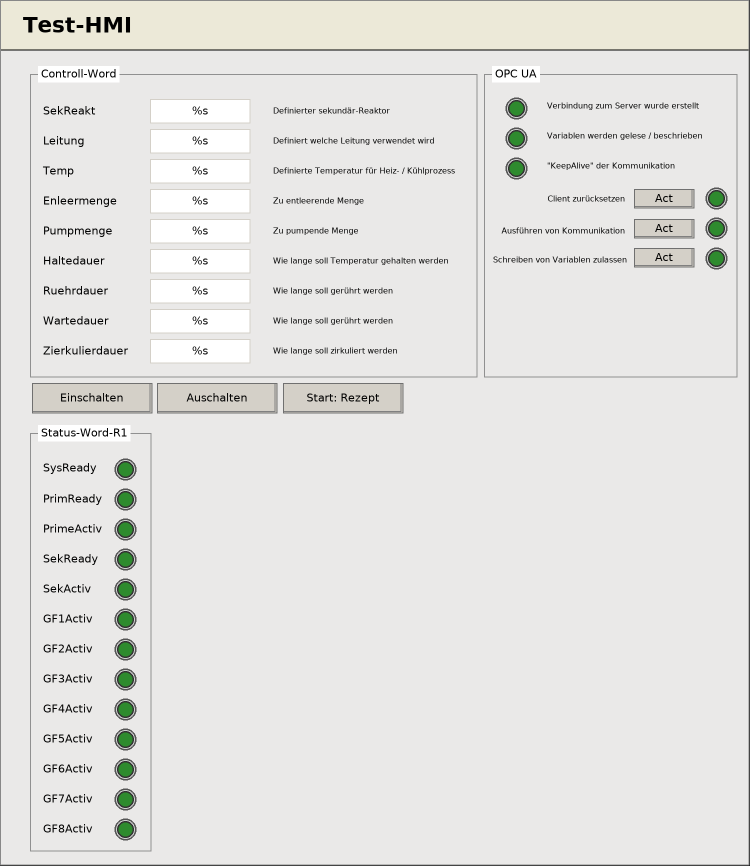
VISUALIZATION Test_Visu  // 750x866
    Rectangle (0,6 750x860)
    Rectangle (0,0 750x50)
    Label (20,0 480x50), "Test-HMI"
    GroupBox (30,66 447x311), "Controll-Word"
        Label (10,30 150x30), "SekReakt"
        Label (10,60 150x30), "Leitung"
        Label (10,90 150x30), "Temp"
        Label (10,120 150x30), "Enleermenge"
        Label (10,150 150x30), "Pumpmenge"
        Label (10,180 150x30), "Haltedauer"
        Label (10,210 150x30), "Ruehrdauer"
        Label (10,240 150x30), "Wartedauer"
        Label (10,270 150x30), "Zierkulierdauer"
        Textfield (120,33 100x24), "%s", text variable: GVL.Param_CW.SekReakt
            OnMouseClick: write GVL.Param_CW.SekReakt via Edit
        Textfield (120,63 100x24), "%s", text variable: GVL.Param_CW.Leitung
            OnMouseClick: write GVL.Param_CW.Leitung via Edit
        Textfield (120,93 100x24), "%s", text variable: GVL.Param_CW.Temp
            OnMouseClick: write GVL.Param_CW.Temp via Edit
        Textfield (120,123 100x24), "%s", text variable: GVL.Param_CW.Enlteermenge
            OnMouseClick: write GVL.Param_CW.Enlteermenge via Edit
        Textfield (120,153 100x24), "%s", text variable: GVL.Param_CW.Pumpmenge
            OnMouseClick: write GVL.Param_CW.Pumpmenge via Edit
        Textfield (120,183 100x24), "%s", text variable: GVL.Param_CW.Haltedauer
            OnMouseClick: write GVL.Param_CW.Haltedauer via Edit
        Textfield (120,213 100x24), "%s", text variable: GVL.Param_CW.Ruehrdauer
            OnMouseClick: write GVL.Param_CW.Ruehrdauer via Edit
        Textfield (120,243 100x24), "%s", text variable: GVL.Param_CW.Wartedauer
            OnMouseClick: write GVL.Param_CW.Wartedauer via Edit
        Textfield (120,273 100x24), "%s", text variable: GVL.Param_CW.Zirkulierdauer
            OnMouseClick: write GVL.Param_CW.Zirkulierdauer via Edit
        Label (240,30 300x30), "Definierter sekundär-Reaktor"
        Label (240,60 300x30), "Definiert welche Leitung verwendet wird"
        Label (240,90 300x30), "Definierte Temperatur für Heiz- / Kühlprozess"
        Label (240,120 300x30), "Zu entleerende Menge"
        Label (240,150 300x30), "Zu pumpende Menge"
        Label (240,180 300x30), "Wie lange soll Temperatur gehalten werden"
        Label (240,210 300x30), "Wie lange soll gerührt werden"
        Label (240,240 300x30), "Wie lange soll gerührt werden"
        Label (240,270 300x30), "Wie lange soll zirkuliert werden"
    GroupBox (30,425 121x426), "Status-Word-R1"
        Label (10,59 150x30), "PrimReady"
        Label (10,89 150x30), "PrimeActiv"
        Label (10,119 150x30), "SekReady"
        Label (10,149 150x30), "SekActiv"
        Label (10,179 150x30), "GF1Activ"
        Label (10,209 150x30), "GF2Activ"
        Label (10,239 150x30), "GF3Activ"
        Label (10,269 150x30), "GF4Activ"
        Label (10,299 150x30), "GF5Activ"
        Label (10,329 150x30), "GF6Activ"
        Label (10,359 150x30), "GF7Activ"
        Label (10,389 150x30), "GF8Activ"
        Lamp1 (83,62 25x25), variable: GVL_OPC_UA.SysSW_R1.GF8Activ, style: Lamp-Lamp1-Green
        Lamp1 (83,92 25x25), variable: GVL_OPC_UA.SysSW_R1.PrimActiv, style: Lamp-Lamp1-Green
        Lamp1 (83,122 25x25), variable: GVL_OPC_UA.SysSW_R1.SekReady, style: Lamp-Lamp1-Green
        Lamp1 (83,152 25x25), variable: GVL_OPC_UA.SysSW_R1.SekActiv, style: Lamp-Lamp1-Green
        Lamp1 (83,182 25x25), variable: GVL_OPC_UA.SysSW_R1.GF1Activ, style: Lamp-Lamp1-Green
        Lamp1 (83,212 25x25), variable: GVL_OPC_UA.SysSW_R1.GF2Activ, style: Lamp-Lamp1-Green
        Lamp1 (83,242 25x25), variable: GVL_OPC_UA.SysSW_R1.GF3Activ, style: Lamp-Lamp1-Green
        Lamp1 (83,272 25x25), variable: GVL_OPC_UA.SysSW_R1.GF4Activ, style: Lamp-Lamp1-Green
        Lamp1 (83,302 25x25), variable: GVL_OPC_UA.SysSW_R1.GF5Activ, style: Lamp-Lamp1-Green
        Lamp1 (83,332 25x25), variable: GVL_OPC_UA.SysSW_R1.GF6Activ, style: Lamp-Lamp1-Green
        Lamp1 (83,362 25x25), variable: GVL_OPC_UA.SysSW_R1.GF7Activ, style: Lamp-Lamp1-Green
        Lamp1 (83,392 25x25), variable: GVL_OPC_UA.SysSW_R1.GF8Activ, style: Lamp-Lamp1-Green
        Lamp1 (83,32 25x25), variable: GVL_OPC_UA.SysSW_R1.GF8Activ, style: Lamp-Lamp1-Green
    Button (283,383 120x30), "Start: Rezept"
        tap GVL.Start
    Button (32,383 120x30), "Einschalten"
        tap GVL.Start
        OnMouseClick: execute { Reaktoranlage.R1.M_M_ON(); }
    Button (157,383 120x30), "Auschalten"
        tap GVL.Start
        OnMouseClick: execute { Reaktoranlage.R1.M_M_OFF(); }
    GroupBox (484,66 253x311), "OPC UA"
        Lamp1 (20,30 25x25), variable: bWrite_Enable, style: Lamp-Lamp1-Green
        Lamp1 (20,60 25x25), variable: bReadBusy, style: Lamp-Lamp1-Green
        Lamp1 (20,90 25x25), variable: bKeepAlives, style: Lamp-Lamp1-Green
        Lamp1 (220,120 25x25), variable: bResetStm, style: Lamp-Lamp1-Green
        Lamp1 (220,150 25x25), variable: bExecute, style: Lamp-Lamp1-Green
        Lamp1 (220,180 25x25), variable: bWrite_Enable, style: Lamp-Lamp1-Green
        Label (60,25 150x30), "Verbindung zum Server wurde erstellt"
        Label (60,55 183x30), "Variablen werden gelese / beschrieben"
        Label (60,85 183x30), ""KeepAlive" der Kommunikation"
        Button (150,123 60x19), "Act"
            tap GVL.Start
            toggle bResetStm
        Button (150,153 60x19), "Act"
            tap GVL.Start
            toggle bExecute
        Button (150,182 60x19), "Act"
            tap GVL.Start
            toggle bWrite_Enable
    Label (445,184 183x30), "Client zurücksetzen"
    Label (445,216 183x30), "Ausführen von Kommunikation"
    Label (447,245 183x30), "Schreiben von Variablen zulassen"
    Label (40,453 150x30), "SysReady"
END_VISUALIZATION

(* stored: Version 1.1.0.1, ProductVersion 3.1.4024.12
   Visu Test_Visu: Id {7a330c66-7157-42cd-ab8d-492a196e9bcc} *)
